{attribute addProperty BoxType "EL9210-0000-0016"}
{attribute addProperty Id "FuseErrorAT %I*BOOL81"}
{attribute addProperty CRC "1047352275"}
{attribute addProperty SizeInBites "8"}
{attribute addProperty SizeInBytes "1"}
TYPE FuseError_3E6D53D3 :
STRUCT
	{attribute addProperty Name "FuseError"}
	FuseError AT %I* : BOOL;
END_STRUCT
END_TYPE

(* stored: Version 1.2.0.0, ProductVersion 3.1.4024.9
   DUT FuseError_3E6D53D3: Id {d606e389-4f4d-4071-8f78-e1e750e0cf19} *)
